Fanuc KAREL source: kb00112.KL

-- PROVISIONAL review KL for V940-1; original PC SHA256 b4ca1b4dd824eb289f7cbb735dd3d0dad2d16089716f54ea75d2f66ab22eba22
-- Incomplete behavior may be omitted. Consult companion uncertainty JSON. Do not deploy.
PROGRAM KB00112
%NOLOCKGROUP
VAR
  RESULT : BOOLEAN
-- UNRESOLVED_DECL P1 type=000199
BEGIN
  -- V9_ZERO_TABLE_METADATA_HINT layout=0001; no indexed target words; source/name/runtime held
  -- UNRESOLVED_PC offsets 5-28; opcodes 27,22,1C,27,9D,76,23
  -- UNRESOLVED_PC offsets 33-37; opcodes 7F
END KB00112
